FUNCTION_BLOCK FB_Axis_HomeToMotorToque EXTENDS FB_Axis_HomeToHardStop
VAR_INPUT
END_VAR
VAR_OUTPUT
END_VAR
VAR
END_VAR

METHOD HardwareUpdate : BOOL
VAR_INPUT
END_VAR
//nTorqueFeedback := SelectedAxis.NcToPlc.ActTorque / ;
END_METHOD

END_FUNCTION_BLOCK

(* stored: Version 1.1.0.1, ProductVersion 3.1.4024.9
   POU FB_Axis_HomeToMotorToque: Id {9379d647-c9c4-4902-85f9-9d975d66d894}, SpecialFunc None
   Folder 01_SUPER_Overrides: Id {4daa08ef-b23d-49f5-8ecb-9bf0e97db98c}
   Method HardwareUpdate: Id {96956867-482c-426e-a993-144b55dd7964} *)
